// TIA Portal V15.1 export
// export: Created 2024-05-17T05:38:25.6668141Z, ExportSetting WithDefaults, DisplayName Totally Integrated Automation Portal, DisplayVersion V15.1 Update 5, DisplayName TIA Portal Openness, DisplayVersion V15.1 Update 5, DisplayName SINAMICS Startdrive Advanced, DisplayVersion V15.1, DisplayName G130, G150, S120, S150, SINAMICS MV, S210, DisplayVersion V15.1, DisplayName G110M, G120, G120C, G120D, G120P, DisplayVersion V15.1, DisplayName STEP 7 Professional, DisplayVersion V15.1 Update 5, DisplayName STEP 7 Safety, DisplayVersion V15.1, DisplayName WinCC Professional, DisplayVersion V15.1 Update 5, DisplayName SIMATIC Visualization Architect, DisplayVersion V15.1
FUNCTION "LModeIAnim" : Void   // FC1006, FBD
TITLE = LModeIAnim
{ S7_Optimized_Access := 'FALSE' }
AUTHOR : VCC
FAMILY : Control
NAME : MIAnim
VERSION : 1.0
// ================================================================================
// Handles the conversion from bits to one Word for a mode icon animation. 
// ================================================================================
// stored: AutoNumber false, IsIECCheckEnabled false, SetENOAutomatically False, UDAEnableTagReadback false
   VAR_INPUT
      I_SetPos : Bool;   // Set position
      I_ResetPos : Bool;   // Reset position
      I_AutoMode : Bool;   // Auto mode
      I_AutoModeSel : Bool;   // Auto selected
      I_StepMode : Bool;   // Step mode
      I_StepModeSel : Bool;   // Step selected
      I_HomeRunMode : Bool;   // Homerun mode
      I_HomeRunModeSel : Bool;   // Homerun selected
      I_ManualMode : Bool;   // Manual mode
      I_ManualModeSel : Bool;   // Manual selected
      I_AnyProdModeActive : Bool;   // Any Production mode active
      I_AnyProdModeSel : Bool;   // Any Production mode sel
      I_AlarmA : Bool;   // AlarmA
      I_AlarmB : Bool;   // AlarmB
      I_AlarmC : Bool;   // AlarmC
      I_AlarmD : Bool;   // AlarmD
   END_VAR
   VAR_OUTPUT
      H_IAnim : Word;   // Icon animation Word
   END_VAR
BEGIN

REGION Network 1: **** 8 - Outputs **** Set position
   // Set position
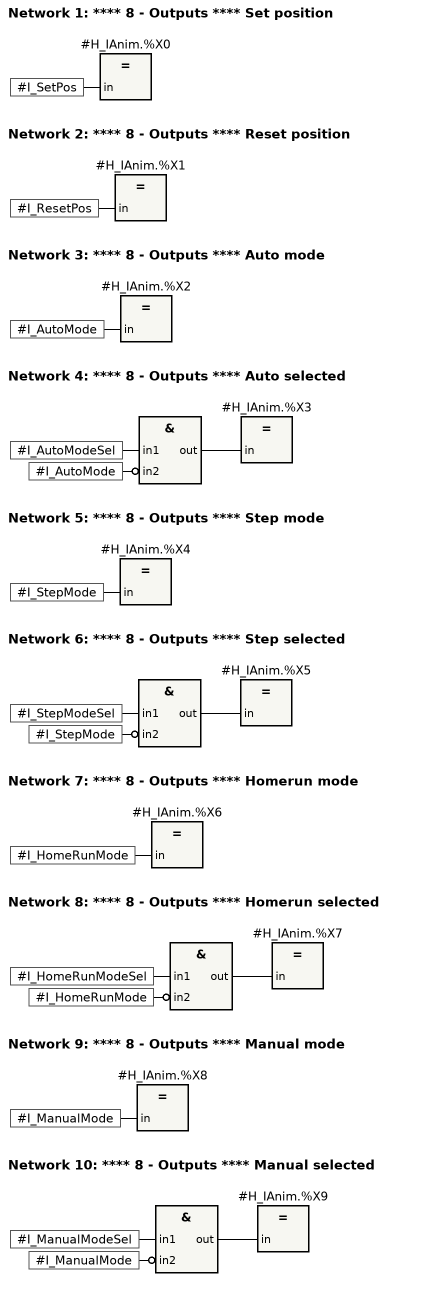
   #H_IAnim.%X0 := #I_SetPos;
END_REGION

REGION Network 2: **** 8 - Outputs **** Reset position
   // Reset position
   #H_IAnim.%X1 := #I_ResetPos;
END_REGION

REGION Network 3: **** 8 - Outputs **** Auto mode
   // Auto mode
   #H_IAnim.%X2 := #I_AutoMode;
END_REGION

REGION Network 4: **** 8 - Outputs **** Auto selected
   // Auto selected
   #H_IAnim.%X3 := #I_AutoModeSel AND NOT #I_AutoMode;
END_REGION

REGION Network 5: **** 8 - Outputs **** Step mode
   // Step mode
   #H_IAnim.%X4 := #I_StepMode;
END_REGION

REGION Network 6: **** 8 - Outputs **** Step selected
   // Step selected
   #H_IAnim.%X5 := #I_StepModeSel AND NOT #I_StepMode;
END_REGION

REGION Network 7: **** 8 - Outputs **** Homerun mode
   // Homerun mode
   #H_IAnim.%X6 := #I_HomeRunMode;
END_REGION

REGION Network 8: **** 8 - Outputs **** Homerun selected
   // Homerun selected
   #H_IAnim.%X7 := #I_HomeRunModeSel AND NOT #I_HomeRunMode;
END_REGION

REGION Network 9: **** 8 - Outputs **** Manual mode
   // Manual mode
   #H_IAnim.%X8 := #I_ManualMode;
END_REGION

REGION Network 10: **** 8 - Outputs **** Manual selected
   // Manual selected
   #H_IAnim.%X9 := #I_ManualModeSel AND NOT #I_ManualMode;
END_REGION

REGION Network 11: **** 8 - Outputs **** Any production mode active
   // Any production mode active
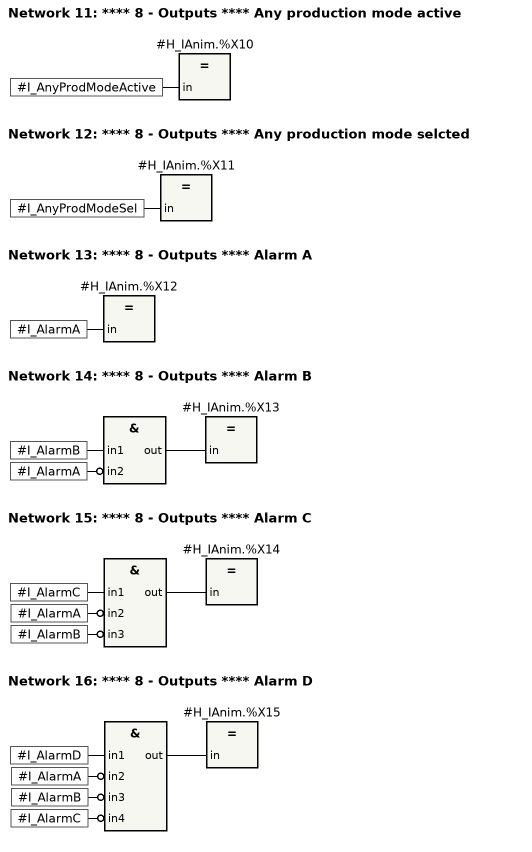
   #H_IAnim.%X10 := #I_AnyProdModeActive;
END_REGION

REGION Network 12: **** 8 - Outputs **** Any production mode selcted
   // Any production mode selcted
   #H_IAnim.%X11 := #I_AnyProdModeSel;
END_REGION

REGION Network 13: **** 8 - Outputs **** Alarm A
   // Alarm A
   #H_IAnim.%X12 := #I_AlarmA;
END_REGION

REGION Network 14: **** 8 - Outputs **** Alarm B
   // Alarm B
   #H_IAnim.%X13 := #I_AlarmB AND NOT #I_AlarmA;
END_REGION

REGION Network 15: **** 8 - Outputs **** Alarm C
   // Alarm C
   #H_IAnim.%X14 := #I_AlarmC AND NOT #I_AlarmA AND NOT #I_AlarmB;
END_REGION

REGION Network 16: **** 8 - Outputs **** Alarm D
   // Alarm D
   #H_IAnim.%X15 := #I_AlarmD AND NOT #I_AlarmA AND NOT #I_AlarmB AND NOT #I_AlarmC;
END_REGION
END_FUNCTION
